{region '#Template'}
	{attribute 'Version' := '5.0.1.0'}
	{attribute 'Tags' := '"LCID": "1031", "Text": "Plant, Weatherstation, Draft"'}
	{attribute 'Tags' := '"LCID": "1033", "Text": "Plant, Weatherstation, Draft"'}
	{attribute 'Using' := '"Type": "Template", "URI": "LblComp"'}		 		 
	{attribute 'Description' := '"LCID": "1031", "Text": "Vorlage-Template: beinhaltet alle Objekte, die Eingangsverknüpfung zu diesen muss vom Anwender erstellt werden"'}
	{attribute 'Description' := '"LCID": "1033", "Text": "Draft-template: contains all objects to be connected to appropriate inputs by the user"'}
{endregion}
FUNCTION_BLOCK FB_BA_WeatherStation_Draft EXTENDS FB_BA_View
VAR_INPUT CONSTANT
	Dstb						: FB_BA_BI;
	Rain						: FB_BA_BI;
	WthT						: FB_BA_AI;
	DewPtT						: FB_BA_AI; 
	PrssAbs						: FB_BA_AI;
	PrssRel						: FB_BA_AI;
	HumAbs						: FB_BA_AI;
	HumRel						: FB_BA_AI;
	Brightness_N				: FB_BA_AI;
	Brightness_S				: FB_BA_AI;
	Brightness_E				: FB_BA_AI;
	Brightness_W				: FB_BA_AI;
	Dawn						: FB_BA_AI;
	GlobRadn					: FB_BA_AI;      
	WndDir						: FB_BA_AI;
	WndSpd						: FB_BA_AI; 
	Latd						: FB_BA_AI;  
	Lngt						: FB_BA_AI; 
	SunAzm						: FB_BA_AI;
	SunElv						: FB_BA_AI;                 
END_VAR	

VAR
	stDateTime_PLACEHOLDER		: TIMESTRUCT;			// Placeholder-variable, so the template can be compiled correctly
														// to be replaced by an appropriate timestruct
END_VAR

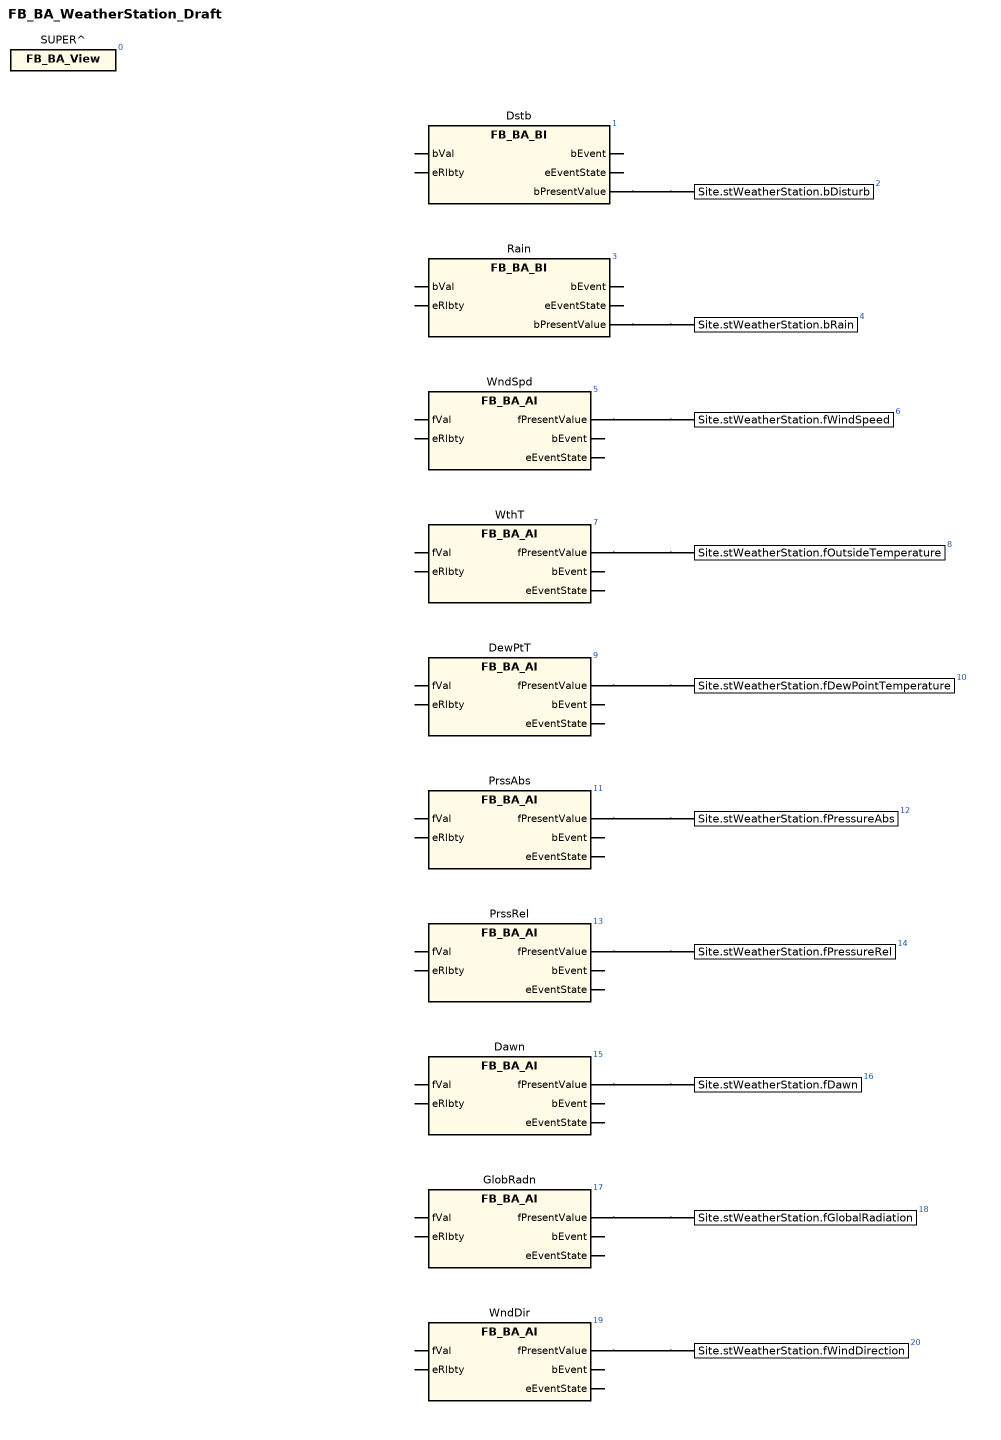
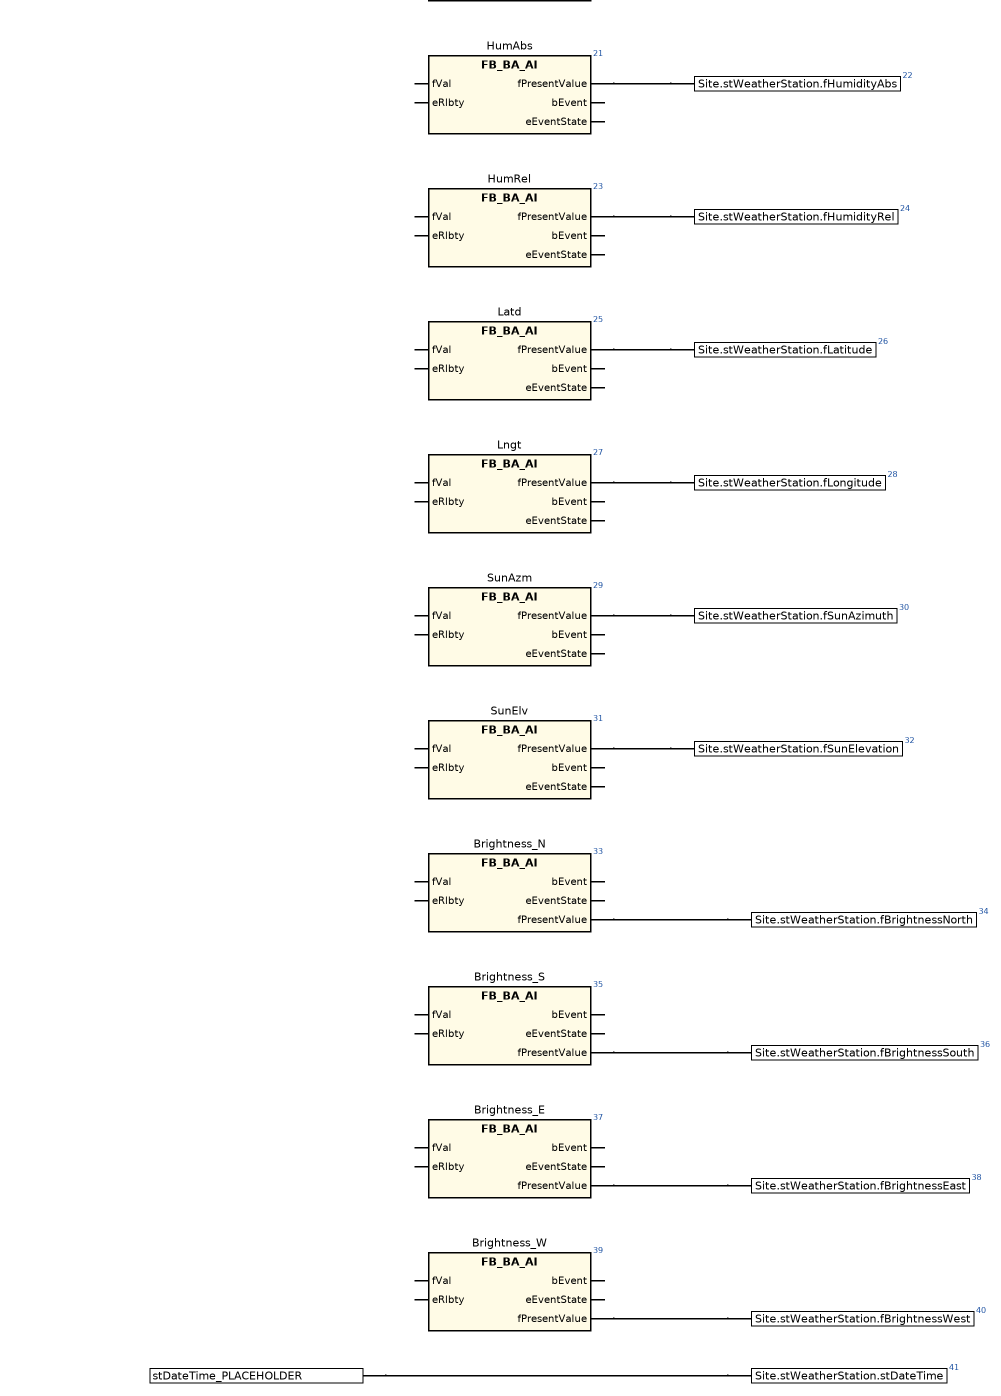
SUPER^(); // FB_BA_View
Dstb(); // FB_BA_BI
Site.stWeatherStation.bDisturb := Dstb.bPresentValue;
Rain(); // FB_BA_BI
Site.stWeatherStation.bRain := Rain.bPresentValue;
WndSpd(); // FB_BA_AI
Site.stWeatherStation.fWindSpeed := WndSpd.fPresentValue;
WthT(); // FB_BA_AI
Site.stWeatherStation.fOutsideTemperature := WthT.fPresentValue;
DewPtT(); // FB_BA_AI
Site.stWeatherStation.fDewPointTemperature := DewPtT.fPresentValue;
PrssAbs(); // FB_BA_AI
Site.stWeatherStation.fPressureAbs := PrssAbs.fPresentValue;
PrssRel(); // FB_BA_AI
Site.stWeatherStation.fPressureRel := PrssRel.fPresentValue;
Dawn(); // FB_BA_AI
Site.stWeatherStation.fDawn := Dawn.fPresentValue;
GlobRadn(); // FB_BA_AI
Site.stWeatherStation.fGlobalRadiation := GlobRadn.fPresentValue;
WndDir(); // FB_BA_AI
Site.stWeatherStation.fWindDirection := WndDir.fPresentValue;
HumAbs(); // FB_BA_AI
Site.stWeatherStation.fHumidityAbs := HumAbs.fPresentValue;
HumRel(); // FB_BA_AI
Site.stWeatherStation.fHumidityRel := HumRel.fPresentValue;
Latd(); // FB_BA_AI
Site.stWeatherStation.fLatitude := Latd.fPresentValue;
Lngt(); // FB_BA_AI
Site.stWeatherStation.fLongitude := Lngt.fPresentValue;
SunAzm(); // FB_BA_AI
Site.stWeatherStation.fSunAzimuth := SunAzm.fPresentValue;
SunElv(); // FB_BA_AI
Site.stWeatherStation.fSunElevation := SunElv.fPresentValue;
Brightness_N(); // FB_BA_AI
Site.stWeatherStation.fBrightnessNorth := Brightness_N.fPresentValue;
Brightness_S(); // FB_BA_AI
Site.stWeatherStation.fBrightnessSouth := Brightness_S.fPresentValue;
Brightness_E(); // FB_BA_AI
Site.stWeatherStation.fBrightnessEast := Brightness_E.fPresentValue;
Brightness_W(); // FB_BA_AI
Site.stWeatherStation.fBrightnessWest := Brightness_W.fPresentValue;
Site.stWeatherStation.stDateTime := stDateTime_PLACEHOLDER;

METHOD FB_init : BOOL
VAR_INPUT
	bInitRetains : BOOL; // if TRUE, the retain variables are initialized (warm start / cold start)
	bInCopyCode : BOOL;  // if TRUE, the instance afterwards gets moved into the copy code (online change)
END_VAR
Dstb.iParent							:= THIS^;
Dstb.iLabel								:= LblComp_Wth_WeatherStation; 	
Dstb.sActiveText 						:= txtEvent_Yes;
Dstb.sInactiveText 						:= txtEvent_No;
Dstb.nEventClassID						:= EC_ID.NC60;
Dstb.aEventTransitionText[1]			:= txtEvent_No;
Dstb.aEventTransitionText[2]			:= txtEvent_None;
Dstb.aEventTransitionText[3]			:= txtEvent_Yes;
Dstb.bEventDetectionEnable				:= FALSE;	  
						
Rain.iParent							:= THIS^;
Rain.iLabel								:= LblComp_Wth_RainSensor; 	
Rain.sActiveText 						:= txtEvent_Yes;
Rain.sInactiveText 						:= txtEvent_No;
Rain.nEventClassID						:= EC_ID.NC60;
Rain.aEventTransitionText[1]			:= txtEvent_No;
Rain.aEventTransitionText[2]			:= txtEvent_None;
Rain.aEventTransitionText[3]			:= txtEvent_Yes;
Rain.bEventDetectionEnable				:= FALSE;	
						
WthT.iParent							:= THIS^;
WthT.iLabel								:= LblComp_Wth_TemperatureOutside; 	
WthT.eUnit 								:= E_BA_Unit.eTemperature_DegreesCelsius;	
WthT.nEventClassID						:= EC_ID.NC40;
										
DewPtT.iParent							:= THIS^;
DewPtT.iLabel							:= LblComp_Wth_TemperatureDewPoint; 		
DewPtT.eUnit							:= E_BA_Unit.eTemperature_DegreesCelsius;
DewPtT.nEventClassID					:= EC_ID.NC40;
						
PrssAbs.iParent							:= THIS^;
PrssAbs.iLabel							:= LblComp_Wth_PressureAbsolute; 
PrssAbs.eUnit							:= E_BA_Unit.ePressure_Hectopascals;
PrssAbs.nEventClassID					:= EC_ID.NC40;
										
PrssRel.iParent							:= THIS^;
PrssRel.iLabel							:= LblComp_Wth_PressureRelative; 	
PrssRel.eUnit							:= E_BA_Unit.ePressure_Hectopascals;
PrssRel.nEventClassID					:= EC_ID.NC40;
						
HumAbs.iParent							:= THIS^;
HumAbs.iLabel							:= LblComp_Wth_AbsoluteHumidityOutsideAir; 
HumAbs.eUnit							:= E_BA_Unit.eHumidity_GramsOfWaterPerKilogramDryAir;
HumAbs.nEventClassID					:= EC_ID.NC40;
										
HumRel.iParent							:= THIS^;
HumRel.iLabel							:= LblComp_Wth_RelativeHumidityOutsideAir; 
HumRel.eUnit							:= E_BA_Unit.eHumidity_PercentRelativeHumidity;
HumRel.nEventClassID					:= EC_ID.NC40;
						
Brightness_N.iParent					:= THIS^;
Brightness_N.iLabel						:= LblComp_Wth_Brightness; 		
Brightness_N.eUnit						:= E_BA_Unit.eLight_Luxes;
Brightness_N.nEventClassID				:= EC_ID.NC40;
                                        
Brightness_S.iParent					:= THIS^;
Brightness_S.iLabel						:= LblComp_Wth_Brightness; 		
Brightness_S.eUnit						:= E_BA_Unit.eLight_Luxes;
Brightness_S.nEventClassID				:= EC_ID.NC40;
                                        
Brightness_E.iParent					:= THIS^;
Brightness_E.iLabel						:= LblComp_Wth_Brightness; 		
Brightness_E.eUnit						:= E_BA_Unit.eLight_Luxes;
Brightness_E.nEventClassID				:= EC_ID.NC40;
                                        
Brightness_W.iParent					:= THIS^;
Brightness_W.iLabel						:= LblComp_Wth_Brightness; 		
Brightness_W.eUnit						:= E_BA_Unit.eLight_Luxes;
Brightness_W.nEventClassID				:= EC_ID.NC40;

Dawn.iParent							:= THIS^;
Dawn.iLabel								:= LblComp_Wth_Dawn; 	
Dawn.eUnit								:= E_BA_Unit.eLight_Luxes;
Dawn.nEventClassID						:= EC_ID.NC40;
						
GlobRadn.iParent						:= THIS^;
GlobRadn.iLabel							:= LblComp_Wth_SolarRadiation; 	
GlobRadn.eUnit							:= E_BA_Unit.eLight_WattsPerSquareMeter;
GlobRadn.nEventClassID					:= EC_ID.NC40;
						
WndDir.iParent							:= THIS^;
WndDir.iLabel							:= LblComp_Wth_WindDirection; 	
WndDir.eUnit							:= E_BA_Unit.eOther_DegreesAngular;
WndDir.nEventClassID					:= EC_ID.NC40;
										
WndSpd.iParent							:= THIS^;
WndSpd.iLabel							:= LblComp_Wth_WindSpeed; 	
WndSpd.eUnit							:= E_BA_Unit.eVelocity_MetersPerSecond;
WndSpd.nEventClassID					:= EC_ID.NC40;
						
Latd.iParent							:= THIS^;
Latd.iLabel								:= LblComp_Wth_GeoLatitude; 	
Latd.eUnit								:= E_BA_Unit.eOther_DegreesAngular;
Latd.nEventClassID						:= EC_ID.NC40;
										
Lngt.iParent							:= THIS^;
Lngt.iLabel								:= LblComp_Wth_GeoLongitude; 	
Lngt.eUnit								:= E_BA_Unit.eOther_DegreesAngular;
Lngt.nEventClassID						:= EC_ID.NC40;
						
SunAzm.iParent							:= THIS^;
SunAzm.iLabel							:= LblComp_Wth_SunAzimuth; 	
SunAzm.eUnit							:= E_BA_Unit.eOther_DegreesAngular;
SunAzm.nEventClassID					:= EC_ID.NC40;
						
SunElv.iParent							:= THIS^;
SunElv.iLabel							:= LblComp_Wth_SunElevation; 	
SunElv.eUnit							:= E_BA_Unit.eOther_DegreesAngular;
SunElv.nEventClassID					:= EC_ID.NC40;
END_METHOD

END_FUNCTION_BLOCK

(* stored: Version 1.1.0.1, ProductVersion 3.1.4024.12
   POU FB_BA_WeatherStation_Draft: Id {468f09d2-8316-4c52-8a17-1f33e2134d15}, SpecialFunc None
   Method FB_init: Id {375ae77a-6d85-4803-b069-11951a6d3132} *)
